FUNCTION BandLimit : LREAL
VAR_INPUT
	Value: LREAL;
	Target: LREAL;
	Width: LREAL;
	MinValue: LREAL;
	MaxValue: LREAL;
END_VAR
VAR
END_VAR

BandLimit := LimitValue(Band(Value, Target, Width), MinValue, MaxValue);

END_FUNCTION

(* stored: Version 1.1.0.1, ProductVersion 3.1.4024.3
   POU BandLimit: Id {0bd8d519-40a2-4181-be9a-2724cdd75315}, SpecialFunc None *)
